TYPE (* IEC61131-3, Table 14#5 *)
  (* Standard: 1131-3 *)
  (* Version 0.0, 8/22/2023, valeriy, nxtControl GmBH, Template *)
  PACKAGE Main;
  DataType1 : STRUCT
    item1 : BOOL;
    item2 : REAL;
    item3 : STRING;
  END_STRUCT;
END_TYPE
